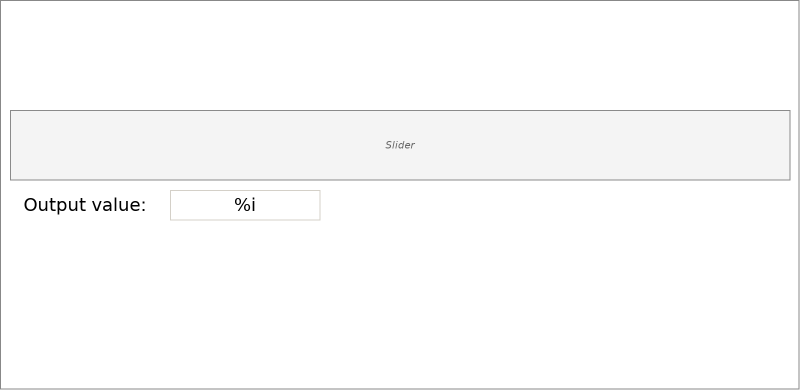
VISUALIZATION VisuAnalogOutControl  // 800x390
VAR_IN_OUT
	fbManualControler	: FB_ManualController ;
END_VAR
    Slider (10,110 780x70), variable: fbManualControler.pDevAnalogOut^.fCmdValue, scale 0..100
    Textfield (170,190 150x30), "%i", text variable: fbManualControler.pDevAnalogOut^.fCmdValue
        OnMouseClick: write the text variable via VisuDialogs.Numpad
    Label (10,190 150x30), "Output value:"
END_VISUALIZATION

(* stored: Version 1.1.0.1, ProductVersion 3.1.4024.9
   Visu VisuAnalogOutControl: Id {6054b02d-98e9-4d8c-9154-935e2b6b306b} *)
